{attribute 'qualified_only'}
{attribute 'strict'}
TYPE ST_SF3_3_RESTART_PREVENTION_EXP :
STRUCT
    bSI_RESET_EXP : BOOL;
    bSI_PSS_ACCESS : BOOL;
END_STRUCT
END_TYPE

(* stored: Version 1.1.0.1
   DUT ST_SF3_3_RESTART_PREVENTION_EXP: Id {a46a440a-a956-0527-0f0f-fdc0940ba3a1} *)
